PROGRAM MAIN
VAR
	v : INT := 0;
END_VAR

v := v+1;
PROG_ReadStructure();

END_PROGRAM

(* stored: Version 1.1.0.1, ProductVersion 3.1.4022.9
   POU MAIN: Id {34399180-6f2e-4cbd-9a60-f52d30bd70e9}, SpecialFunc None *)
